ABB RAPID module: TCPZ_boor_11mm_280lang.mod

MODULE TCPZ_boor_11mm_280lang
	! Points are read in order of declaration.
  ! Please do not change the order of points!

  LOCAL PERS robtarget pTCPZ_Point1:=[[565.2722,-1599.526,937.3368],[0.236160889267921,0.602700293064117,0.212920904159546,-0.731877744197845],[-1,0,-1,0],[9E+09,9E+09,9E+09,9E+09,9E+09,9E+09]];
	LOCAL PERS robtarget pTCPZ_Point2:=[[127.5661,-1689.504,917.5461],[0.227667048573494,0.852620899677277,0.147526755928993,-0.446588307619095],[-1,1,-1,0],[9E+09,9E+09,9E+09,9E+09,9E+09,9E+09]];
	LOCAL PERS robtarget pTCPZ_Point3:=[[265.8278,-1380.54,860.8713],[0.712427496910095,0.227243512868881,0.485931903123856,-0.452413141727448],[-1,-1,0,0],[9E+09,9E+09,9E+09,9E+09,9E+09,9E+09]];
	LOCAL PERS robtarget pTCPZ_Point4:=[[386.6405,-1609.824,966.8923],[0.499783664941788,0.500724911689758,0.499924302101135,-0.499566316604614],[-1,0,-1,0],[9E+09,9E+09,9E+09,9E+09,9E+09,9E+09]];
	LOCAL PERS robtarget pTCPZ_ElongZ:=[[386.6398,-1609.823,1154.507],[0.499783426523209,0.500726342201233,0.499924957752228,-0.499564468860626],[-1,0,-1,0],[9E+09,9E+09,9E+09,9E+09,9E+09,9E+09]];

ENDMODULE
